RoboDK station: Final_preparion_gripper.rdk

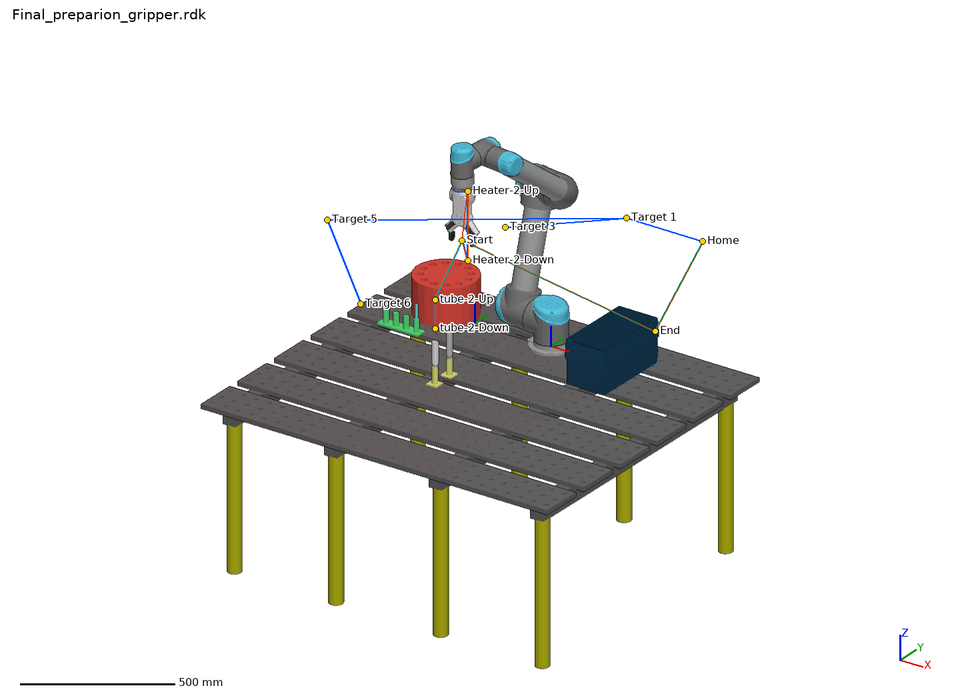
[picture v0: the station drawn from its stored meshes, robots at their saved joint values, targets as dots, program paths as lines]
Station Final_preparion_gripper (saved by RoboDK 5.3.4). Poses are relative to the parent item; angles as X-Y-Z fixed-axis rotations.
Station parameters (name, value as stored): IO_5, 1, IO_16, 0, IO_17, 1, IO_11, 1, IO_18, 1, IO_10, 0
  - frame World at (-300, 0, 0) mm
    - object Table at (0, 0, 0) mm, size 1193.8 x 965.2 x 609.6 mm, geometry from welding_table.sld
    - object Heater at (0, 0, 0) mm, size 225 x 140 x 222.7 mm, geometry from Heater.stl
    - object SFixture_2 at (0, 0, 0) mm, size 160 x 40 x 50 mm, geometry from Fixture_2.stp
    - object Smalltube at (0, 0, 0) mm, size 12 x 12 x 100 mm, geometry from Smalltube.stp
    - object Fixture_1 at (0, 0, 0) mm, size 40 x 63 x 40 mm, geometry from Fixture_1.stl
    - object Test-tube-1 at (0, 0, 0) mm, size 22 x 147.5 x 22 mm, geometry from Test-tube.stl
    - object Fixture_2 at (0, 0, 0) mm, size 40 x 63 x 40 mm, geometry from Fixture_1.stl
    - object Test-tube-2 at (0, 0, 0) mm, size 22 x 147.5 x 22 mm, geometry from Test-tube.stl
    - object Waterbox at (0, 0, 0) mm, size 166 x 315.8 x 161.6 mm, geometry from Box-400mmx200mm-Opened.sld
    - object Table_2 at (0, 0, 0) mm, size 1193.8 x 965.2 x 609.6 mm, geometry from welding_table.sld
  - frame Working at (-300, 0, 0) mm
    - target tube-2-Up (Cartesian target) at (-147.01, -443.12, 302.87) mm, rotated rx 180 ry 0.01 rz 90 deg; joints [-94.853, -86.546, -82.967, -100.477, 90.001, 85.147] of UR5
    - target tube-2-Down (Cartesian target) at (-147.01, -443.14, 199.34) mm, rotated rx 180 ry 0.01 rz 90 deg; joints [-94.853, -85.837, -98.805, -85.348, 90.001, 85.147] of UR5
    - target Heater-2-Down (Cartesian target) at (-339.09, 16.37, 205.17) mm, rotated rx 179.99 ry 0 rz -2.65 deg; joints [-164.045, -67.225, -111.884, -90.888, 90.01, 108.602] of UR5
    - target Heater-2-Up (Cartesian target) at (-339.09, 16.37, 455) mm, rotated rx 179.99 ry 0 rz -2.65 deg; joints [-164.045, -77.973, -65.763, -126.261, 90.01, 108.602] of UR5
  - frame UR5 Base at (-300, 0, 0) mm
    - robot UR5: 6 axes, payload 5 kg, reach 850 mm, repeatability 0.1 mm, weight 18.4 kg
        modified DH rows (alpha deg, a mm, theta deg, d mm): 0, 0, 0, 89.2; 90, 0, 180, 0; 0, 425, 0, 0; 0, 392.43, 0, 109; -90, 0, 0, 93.65; 90, 0, 180, 82
        joint limits [-360, -360, -360, -360, -360, -360] to [360, 360, 360, 360, 360, 360]; home [0, -90, -90, 0, 90, 0]; saved at [-97.276, -76.28, -66.912, -126.799, 90.001, 82.724]
      - tool RG2_v2, TCP at (0, 0, 200) mm, size 211.5 x 123 x 75.3 mm, geometry from RG2_v2.STEP
  - frame Calibration Target at (-300, 0, 0) mm
    - target Home (Cartesian target) at (674.43, -109, 607.85) mm, rotated rx -90 ry 0 rz -90 deg; joints [0, -90, -90, 0, 90, 0] of UR5
    - target End (Cartesian target) at (486.13, -109, 232.28) mm, rotated rx -179.99 ry 0 rz -90 deg; joints [0, -90, -89.99, -90, 90, 0] of UR5
    - frame Test at (-300, 0, 0) mm
      - target Target 1 (Cartesian target) at (674.43, -109, 607.85) mm, rotated rx 0 ry 90 rz 0 deg; joints [0, -90, -90, 0, 90, 90] of UR5
      - target Target 2 (Cartesian target) at (674.43, -109, 607.85) mm, rotated rx 0 ry -90 rz 180 deg; joints [0, -90, -90, 0, 90, -90] of UR5
      - target Target 3 (Cartesian target) at (392.43, -391, 607.85) mm, rotated rx 0 ry -90 rz 90 deg; joints [0, -90, -90, 0, 0, -90] of UR5
      - target Target 4 (Cartesian target) at (674.43, -109, 607.85) mm, rotated rx 0 ry -90 rz 180 deg; joints [0, -90, -90, 0, 90, -90] of UR5
      - target Target 5 (Cartesian target) at (-109, -674.43, 607.85) mm, rotated rx 0 ry -90 rz 90 deg; joints [-90, -90, -90, 0, 90, -90] of UR5
      - target Target 6 (Cartesian target) at (-109, -486.08, 232.2) mm, rotated rx 180 ry 0 rz -90 deg; joints [-90, -90, -90, -90, 90, -90] of UR5
    - target Start (Cartesian target) at (-147.01, -290.81, 455.21) mm, rotated rx 180 ry 0.01 rz 90 deg; joints [-97.276, -76.28, -66.912, -126.799, 90.001, 82.724] of UR5
  - program Calibration (13 instructions, listed below)
  - program Move to start point (7 instructions, listed below)
  - program Back to home (6 instructions, listed below)
  - Python program Open_the_gripper (listed below)
  - Python program Close_the_gripper (listed below)
  - Python program rInitial (listed below)
  - program MainProgram (4 instructions, listed below)
  - program Back to start (4 instructions, listed below)
  - program Open_the _gripper (1 instructions, listed below)
  - program Close_the_gripper (1 instructions, listed below)
  - program Pickup tube2 prepared (10 instructions, listed below)
  - program Back from 2 (7 instructions, listed below)
  - program Place tube2 prepared  (8 instructions, listed below)
  - program MP_Pickup 2 from 2 (4 instructions, listed below)
  - program MP_Place 2 to 2 (4 instructions, listed below)
  - program PY_MainProgram (4 instructions, listed below)
  - program Pickup from heater_1 (10 instructions, listed below)
  - program Place to heater_2 (11 instructions, listed below)
  - program MP_H2_to_F2 (3 instructions, listed below)
  - program MP_F2_to_H2 (3 instructions, listed below)
  - program MainProgram (7 instructions, listed below)
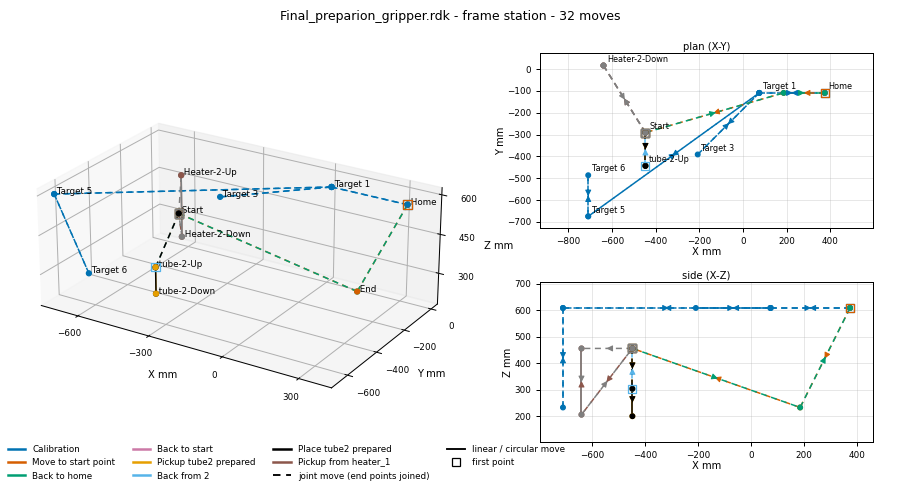
[picture p0: tool path of Final_preparion_gripper.rdk in frame station, 32 of 32 moves have a stored position in this frame; points joined in program order, loops and branches not executed]

--- program Calibration (robot UR5) ---
  替换物体
  设置参考: Calibration -> Calibration Target
  设置工具: RG2_v2
  MoveJ (Home)
  MoveJ (Target 1)
  MoveJ (Target 2)
  MoveJ (Target 3)
  MoveJ (Target 4)
  MoveJ (Target 5)
  MoveJ (Target 6)
  MoveJ (Target 5)
  MoveJ (Target 4)
  MoveJ (Home)

--- program Move to start point (robot UR5) ---
  替换物体
  设置参考: Calibration Target
  设置工具: RG2_v2
  设置速度（100.0 mm/s)
  MoveJ (Home)
  MoveJ (End)
  MoveJ (Start)

--- program Back to home (robot UR5) ---
  替换物体
  设置参考: Calibration Target
  设置工具: RG2_v2
  MoveJ (Start)
  MoveJ (End)
  MoveJ (Home)

--- Python program Open_the_gripper ---
# Type help("robolink") or help("robodk") for more information
# Press F5 to run the script
# Documentation: https://robodk.com/doc/en/RoboDK-API.html
# Reference:     https://robodk.com/doc/en/PythonAPI/index.html
# Note: It is not required to keep a copy of this file, your python script is saved with the station
from robolink import *    # RoboDK API
from robodk import *      # Robot toolbox
import socket
import time

RDK = Robolink()

# IP-addr/ports for UR
UR_IP = '192.168.0.102'
UR_PORT = 30001



def connect_UR():
    ur_socket = socket.socket(socket.AF_INET, socket.SOCK_STREAM)
    ur_socket.settimeout(2)
    ur_socket.connect((UR_IP, UR_PORT))
    return ur_socket



def send_cmd(ur_socket, cmd):
    cmd = cmd + '\n'
    received=ur_socket.send(cmd.encode())
    received = ur_socket.recvfrom(4096)

    return received



def main():
    ur_socket = connect_UR()
    result = send_cmd(ur_socket, "set_tool_digital_out(0, False)" + "\n")
    time.sleep(1)



if __name__ == "__main__":
    main()

--- Python program Close_the_gripper ---
# Type help("robolink") or help("robodk") for more information
# Press F5 to run the script
# Documentation: https://robodk.com/doc/en/RoboDK-API.html
# Reference:     https://robodk.com/doc/en/PythonAPI/index.html
# Note: It is not required to keep a copy of this file, your python script is saved with the station
from robolink import *    # RoboDK API
from robodk import *      # Robot toolbox
import socket
import time

RDK = Robolink()

# IP-addr/ports for UR
UR_IP = '192.168.0.102'
UR_PORT = 30001



def connect_UR():
    ur_socket = socket.socket(socket.AF_INET, socket.SOCK_STREAM)
    ur_socket.settimeout(2)
    ur_socket.connect((UR_IP, UR_PORT))
    return ur_socket



def send_cmd(ur_socket, cmd):
    cmd = cmd + '\n'
    received=ur_socket.send(cmd.encode())
    received = ur_socket.recvfrom(4096)

    return received



def main():
    ur_socket = connect_UR()
    result = send_cmd(ur_socket, "set_tool_digital_out(0, True)" + "\n")
    time.sleep(1)



if __name__ == "__main__":
    main()

--- Python program rInitial ---
# Type help("robolink") or help("robodk") for more information
# Press F5 to run the script
# Documentation: https://robodk.com/doc/en/RoboDK-API.html
# Reference:     https://robodk.com/doc/en/PythonAPI/index.html
# Note: It is not required to keep a copy of this file, your python script is saved with the station
from robolink import *    # RoboDK API
from robodk import *      # Robot toolbox
import socket
import time
RDK = Robolink()
UR_IP = '192.168.0.102'
UR_PORT = 30001


def connect_UR():
    ur_socket = socket.socket(socket.AF_INET, socket.SOCK_STREAM)
    ur_socket.settimeout(2)
    ur_socket.connect((UR_IP, UR_PORT))
    return ur_socket


def send_cmd(ur_socket, cmd):
    cmd = cmd + '\n'
    received=ur_socket.send(cmd.encode())
    received = ur_socket.recvfrom(4096)
    return received



#ur_socket = connect_UR()
prog = RDK.Item('Back to home', ITEM_TYPE_PROGRAM)
#result = send_cmd(ur_socket, "prog.RunProgram()" + "\n")
#prog = RDK.Item('Back to home', ITEM_TYPE_PROGRAM)
#prog.RunProgram()
RDK.RunProgram('Back to home')
while prog.Busy():
    pause(0.1)
    py_script = RDK.Item('Open_the_gripper')
    py_script.RunProgram()

--- program MainProgram (robot UR5) ---
  Pause 5.0 s
  Call MP_Pickup 2 from 2
  Pause 500 ms
  Call MP_Place 2 to 2

--- program Back to start (robot UR5) ---
  替换物体
  设置参考: Calibration Target
  设置工具: RG2_v2
  MoveJ (Start)

--- program Open_the _gripper (robot UR5) ---
  Set IO_10=0

--- program Close_the_gripper (robot UR5) ---
  Set IO_10=1

--- program Pickup tube2 prepared (robot UR5) ---
  Replace objects
  Set Ref.: Working
  Set Tool: RG2_v2
  Set speed (500.0 mm/s)
  MoveJ (Start)
  Pause 2.5 s
  Call Open_the _gripper
  MoveJ (tube-2-Up)
  Set speed (100.0 mm/s)
  MoveL (Target 2) -> target tube-2-Down

--- program Back from 2 (robot UR5) ---
  Replace objects
  Set Ref.: Working
  Set Tool: RG2_v2
  Set speed (100.0 mm/s)
  MoveL (tube-2-Up)
  Set speed (500.0 mm/s)
  MoveJ (Start)

--- program Place tube2 prepared  (robot UR5) ---
  Replace objects
  Set Ref.: Working
  Set Tool: RG2_v2
  Set speed (500.0 mm/s)
  MoveJ (Start)
  MoveJ (tube-2-Up)
  Set speed (50.0 mm/s)
  MoveL (Target 2) -> target tube-2-Down

--- program MP_Pickup 2 from 2 (robot UR5) ---
  Call Pickup tube2 prepared
  Call Close_the_gripper
  Pause 2.5 s
  Call Back from 2

--- program MP_Place 2 to 2 (robot UR5) ---
  Call Place tube2 prepared
  Call Open_the _gripper
  Pause 2.5 s
  Call Back from 2

--- program PY_MainProgram (robot UR5) ---
  Run Open_the_gripper
  Call Pickup tube2 prepared
  Run Close_the_gripper
  Call Back from 2

--- program Pickup from heater_1 (robot UR5) ---
  Replace objects
  Set Ref.: Calibration Target
  Set Tool: RG2_v2
  Set speed (500.0 mm/s)
  MoveJ (Start)
  MoveJ (Heater-2-Down)
  Call Close_the_gripper
  Pause 2.5 s
  Set speed (50.0 mm/s)
  MoveL (Heater-2-Up)

--- program Place to heater_2 (robot UR5) ---
  Replace objects
  Set Ref.: Working
  Set Tool: RG2_v2
  Set speed (200.0 mm/s)
  MoveJ (Start)
  MoveJ (Heater-2-Up)
  Set speed (50.0 mm/s)
  MoveL (Heater-2-Down)
  Call Open_the _gripper
  Pause 2.5 s
  MoveJ (Start)

--- program MP_H2_to_F2 (robot UR5) ---
  Call Pickup from heater_1
  Pause 500 ms
  Call MP_Place 2 to 2

--- program MP_F2_to_H2 (robot UR5) ---
  Call MP_Pickup 2 from 2
  Pause 500 ms
  Call Place to heater_2

--- program MainProgram (robot UR5) ---
  Pause 2.5 s
  Call Open_the _gripper
  Call MP_F2_to_H2
  Pause 1.5 s
  Call MP_H2_to_F2
  Call Close_the_gripper
  Call Back to home
